KUKA KRL data list: A04_swp_global.dat

&ACCESS RV
&COMMENT V_1_4_0
DEFDAT A04_swp_global PUBLIC
;********************************
;Date: 20.12.2013
;Programmer: GG (KUKA Roboter GmbH)
;Description: Global positions
;********************************
ENDDAT
